DATA_BLOCK "DB"
{ S7_Optimized_Access := 'false' }
    VAR
        aut_y: REAL;
        i: DINT;
        bol: BOOL;
        col: BYTE;
        firstRun: BOOL;
    END_VAR
BEGIN
    firstRun := TRUE;
END_DATA_BLOCK
